// TwinCAT 3 PLC project Tank
// ProgramVersion: 3.1.4024.0
// libraries:
//   Tc2_ControllerToolbox, * (Beckhoff Automation GmbH)
//   Tc2_Standard, * (Beckhoff Automation GmbH)
//   Tc2_System, * (Beckhoff Automation GmbH)
//   Tc3_Module, * (Beckhoff Automation GmbH)
// project tree:
//   DUTs/ ST_TankType.TcDUT
//   / PlcTask.TcTTO
//   POUs/ FB_TankSim.TcPOU, MAIN.TcPOU
// real-time tasks:
//   TASK PlcTask: cycle T#10ms, priority 20, ADS port 350

CONFIGURATION Tank
    RESOURCE PLC ON TwinCAT3
        TASK PlcTask(INTERVAL := T#10ms, PRIORITY := 20);
        PROGRAM MAIN WITH PlcTask : MAIN;
    END_RESOURCE
END_CONFIGURATION

// ---- DUTs/ST_TankType.TcDUT
TYPE ST_TankType :
	STRUCT
		h1:REAL;	// Height of liquid 1 in tank 1	[m]
		h2:REAL;	// Height of liquid 1 in tank 2 [m]
		h3:REAL;	// Height of liquid 1 in tank 3 [m]
		k0:REAL;	// Coefficient of input flow
		k1:REAL;	// Coefficient of output flow 1 [m^2/s]
		k2:REAL;	// Coefficient of output flow 2	[m^2/s]
		k3:REAL;	// Coefficient of output flow 3	[m^2/s]
		A1:REAL;	// Area of tank 1	[m^2]
		A2:REAL;	// Area of tank 2	[m^2]
		A3:REAL;	// Area of tank 3	[m^2]
	END_STRUCT
END_TYPE

// ---- POUs/MAIN.TcPOU
PROGRAM MAIN
VAR
	bFirstScan:BOOL := TRUE;
	// Tank Type: Function Block and struct
	StTank:ST_TankType;		// Structured type variable. (intentional St =/= st?)
	rInput:REAL;
	fb_Tank:FB_TankSim;		// Function Block instance. (intentional TankSIM =/= TankSim?)
	
	// PID Instantiation
	fb_PID: FB_CTRL_PID;				// PID instance
	ST_PID_PARAMS:ST_CTRL_PID_PARAMS;	// PID parameters structure
	eMode: E_CTRL_MODE; 				// PID Mode selection

	// PID Function Block inputs
	fSetPointValue : LREAL;
	fActualValue   : LREAL;
	fManSyncValue  : LREAL;
	bSync : BOOL;
	bHold : BOOL; 
END_VAR

IF bFirstScan THEN			// One time initializations
	bFirstScan := FALSE;
	StTank.k0 := 0.1;
	StTank.k1 := 0.2;
	StTank.k2 := 0.25;
	StTank.k3 := 0.3;
	StTank.A1 := 2.0;
	StTank.A2 := 3.0;
	StTank.A3 := 4.0;
	
	st_PID_PARAMS.tTaskCycleTime:= T#10MS; 	// PLC Task Cycle Time
	st_PID_PARAMS.tCtrlCycleTime:= T#10MS;	// Cycle Time of controller >= Task cycle time
	st_PID_PARAMS.fOutMaxLimit:= 5.0;		// Max allowed control output, ORIGINAL 1.0
	st_PID_PARAMS.fOutMinLimit:= 0.0;		// Min allowed control output
	
	fSetpointValue := 0.1;		// SP/reference for height in tank #3
	eMode := eCTRL_MODE_Manual;	// Set the PID control mode to manual
	
	st_PID_PARAMS.fKp :=    8.7775;	// P: Proportional gain
	st_PID_PARAMS.tTn :=  T#18260MS;	// I: Integral time constant (Ti)
	st_PID_PARAMS.tTv :=  T#4565MS;	// D: Derivative time constant (Td)
	st_PID_PARAMS.tTd :=  T#10MS;	// D: filter time constant
	
END_IF

fb_Tank(rU 		:= rInput,	// Call Function Block
		rDeltaT := 0.01,
		StTank  := StTank);
		
fActualValue := StTank.h3;	// Actual value of the height to the controller

// PID call
fb_PID( fSetPointValue := fSetPointValue,
		fActualValue := fActualValue,
		fManSyncValue := fManSyncValue,
		bSync := bSync,
		eMode := eMode,
		bHold := bHold,
		stParams := ST_PID_PARAMS,
		fOut => rInput
	  );

END_PROGRAM

// ---- POUs/FB_TankSim.TcPOU
FUNCTION_BLOCK FB_TankSim
VAR_INPUT
	rU:REAL;
	rDeltaT:REAL;
END_VAR

VAR_IN_OUT
	stTank:ST_TankType;		// Structure, gives needed attributes. (Currently =/= StTank)
END_VAR

VAR_OUTPUT
END_VAR

VAR
	u:REAL;
	h1:REAL;
	h2:REAL;
	h3:REAL;
END_VAR

IF (rU < 0) THEN
	u := 0.0;
ELSIF (u > 1) THEN
	u := 1.0;
ELSE
	u := rU;
END_IF;

// h_k+1 = h_k + dt*(inFlow - outFlow)
h1 := stTank.h1 + rDeltaT*(stTank.k0*u         - stTank.k1*stTank.h1)/stTank.A1;
h2 := stTank.h2 + rDeltaT*(stTank.k1*stTank.h1 - stTank.k2*stTank.h2)/stTank.A2;
h3 := stTank.h3 + rDeltaT*(stTank.k2*stTank.h2 - stTank.k3*stTank.h3)/stTank.A3;

stTank.h1 := h1;
stTank.h2 := h2;
stTank.h3 := h3;

END_FUNCTION_BLOCK
